{attribute 'qualified_only'}
{attribute 'strict'}
TYPE E_EventType :
(
	Alarm := 0,
	Message := 1
);
END_TYPE

(* stored: Version 1.1.0.1, ProductVersion 3.1.4024.9
   DUT E_EventType: Id {97cfa0b0-7cad-4a38-838a-8641c3bc14b0} *)
